{attribute 'OPC.UA.DA' := '1'}
{attribute 'OPC.UA.DA.StructuredType' := '1'}
TYPE SensorTypeMsg :
STRUCT
	Id : EPowerIlluminationFlow;
	SensorType : STRING(255);
END_STRUCT
END_TYPE

(* stored: Version 1.1.0.1, ProductVersion 3.1.4024.10
   DUT SensorTypeMsg: Id {bf1688f0-bbe8-4db6-92d1-2cf64f3aa202} *)
